INTERFACE PUBLIC I_Cyclic EXTENDS __System.IQueryInterface

METHOD PUBLIC CyclicCall
END_METHOD

END_INTERFACE

(* stored: Version 1.1.0.1
   Itf I_Cyclic: Id {29724a98-39fb-49ef-8269-a4963832a6e1}
   Method CyclicCall: Id {c92fe7fa-b2bc-0ca6-2013-379b47cda8d3} *)
